# EPICS StreamDevice protocol: agilent53220ASup/Db/Agilent53220A.proto
#
#
InTerminator  = "\r\n53220A>";
#InTerminator  = "\r\n53210A>";
OutTerminator = CR LF;
ReplyTimeout  =  5000;
ReadTimeout   =  5000;
WriteTimeout  =  10000;
ExtraInput    = Ignore;

# System
GET_IDN             { out "*IDN?";              in "%39c"; }
RESET               { out "*RST";                          }

# Measurement
GET_FREQ            { out "READ?";              in "READ?\r\n%E";}
GET_IMPEDANCE       { out "INP:IMP?";			in "INP:IMP?\r\n%{+1.00000000E+006|+5.00000000E+001}";}
SET_IMPEDANCE       { out "INP:IMP %{1.0E6|50}";in "%*s"; @init{ GET_IMPEDANCE;}}
GET_TRIG_LEVEL      { out "INP:LEV:ABS?";       in "INP:LEV:ABS?\r\n%E";}
SET_TRIG_LEVEL      { out "INP:LEV:ABS %E";     in "%*s"; @init{ GET_TRIG_LEVEL;}}
GET_TRIG_PERCENT    { out "INP:LEV:REL?";       in "INP:LEV:REL?\r\n%d";}
SET_TRIG_PERCENT    { out "INP:LEV:REL %d";     in "%*s"; @init{ GET_TRIG_PERCENT;}}
GET_AUTO_LEVEL      { out "INP:LEV:AUTO?";       in "INP:LEV:AUTO?\r\n%{OFF|ON|ONCE}";}
SET_AUTO_LEVEL      { out "INP:LEV:AUTO %{OFF|ON|ONCE}";     in "%*s"; @init{ GET_AUTO_LEVEL;}}
GET_COUPLING        { out "INP:COUP?";			in "INP:COUP?\r\n%{AC|DC}";}
SET_COUPLING        { out "INP:COUP %{AC|DC}";  in "%*s"; @init{ GET_COUPLING;}}
GET_NOISE_REJ       { out "INP:NREJ?";			in "INP:NREJ?\r\n%{OFF|ON}";}
SET_NOISE_REJ       { out "INP:NREJ %{OFF|ON}";  in "%*s"; @init{ GET_NOISE_REJ;}}
GET_ROSC_SOUR       { out "ROSC:SOUR?";            in "ROSC:SOUR?\r\n%{INT|EXT}";}
SET_ROSC_SOUR       { out "ROSC:SOUR %{INT|EXT}";  in "%*s"; @init{ GET_ROSC_SOUR;}}
GET_ROSC_EXTFREQ    { out "ROSC:EXT:FREQ?";        in "ROSC:EXT:FREQ?\r\n%{+1.00000000E+006|+5.00000000E+006|+1.00000000E+007}";}
SET_ROSC_EXTFREQ    { out "ROSC:EXT:FREQ %{1E6|5E6|10E6}"; in "%*s"; @init{ GET_ROSC_EXTFREQ;}}
GET_DISPDIG_AUTO    { out "DISP:DIG:MASK:AUTO?";        in "DISP:DIG:MASK:AUTO?\r\n%{0|1}";}
SET_DISPDIG_AUTO    { out "DISP:DIG:MASK:AUTO %{OFF|ON}";  in "%*s"; @init{ GET_DISPDIG_AUTO;}}
GET_DISPDIG         { out "DISP:DIG:MASK?";        in "DISP:DIG:MASK?\r\n%d";}
SET_DISPDIG         { out "DISP:DIG:MASK %d";      in "%*s"; @init{ GET_DISPDIG;}}
